// TIA Portal project "移位运算" (V13)

(* hardware
DEVICE "S7300/ET200M station_1"  S7-300 station
   slot 0: "导轨_0"  Rail  6ES7 390-1***0-0AA0
   slot 2: "PLC_1"  CPU 314C-2 PN/DP  6ES7 314-6EH04-0AB0  V3.3
      slot 2: "PROFINET 接口_1"  PN-IO
         slot 1: "Port_1"  Port
         slot 2: "Port_2"  Port
      slot 5: "DI 24/DO 16_1"  DI24/DO16
      slot 6: "AI 5/AO 2_1"  AI5/AO2
      slot 7: "计数_1"  Counter
      slot 8: "定位_1"  Positioning
*)

// ===== PLC "PLC_1"  CPU 314C-2 PN/DP =====

VAR_GLOBAL   // PLC tag table "默认变量表"
   "tag_1" AT %M0.0 : Bool;
   "tag_2" AT %M0.1 : Bool;
   "tag_3" AT %M0.2 : Bool;
   "tag_4" AT %MW100 : Int;
   "tag_5" AT %M0.3 : Bool;
   "tag_6" AT %M0.4 : Bool;
   "tag_7" AT %MW110 : Word;
   "tag_8" AT %MW120 : Word;
   "tag_9" AT %MW130 : Int;
END_VAR

ORGANIZATION_BLOCK "Main"   // OB1, LAD
TITLE = "Main Program Sweep (Cycle)"
{ S7_Optimized_Access := 'FALSE' }
VERSION : 0.1
   VAR_TEMP
      OB1_EV_CLASS : Byte;   // Bits 0-3 = 1 (Coming event), Bits 4-7 = 1 (Event class 1)
      OB1_SCAN_1 : Byte;   // 1 (Cold restart scan 1 of OB 1), 3 (Scan 2-n of OB 1)
      OB1_PRIORITY : Byte;   // Priority of OB Execution
      OB1_OB_NUMBR : Byte;   // 1 (Organization block 1, OB1)
      OB1_RESERVED_1 : Byte;   // Reserved for system
      OB1_RESERVED_2 : Byte;   // Reserved for system
      OB1_PREV_CYCLE : Int;   // Cycle time of previous OB1 scan (milliseconds)
      OB1_MIN_CYCLE : Int;   // Minimum cycle time of OB1 (milliseconds)
      OB1_MAX_CYCLE : Int;   // Maximum cycle time of OB1 (milliseconds)
      OB1_DATE_TIME : Date_And_Time;   // Date and time OB1 started
   END_VAR
BEGIN

REGION Network 1
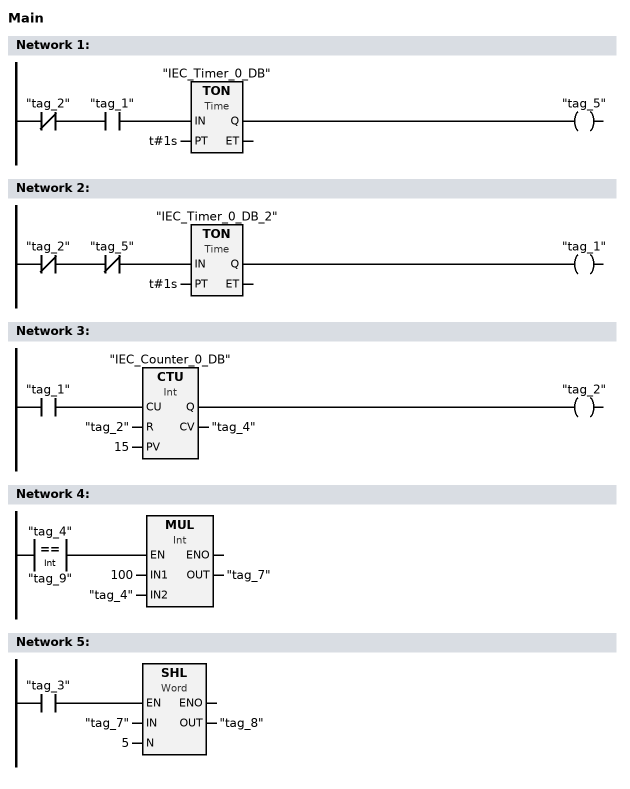
   "IEC_Timer_0_DB".TON(IN := NOT "tag_2" AND "tag_1", PT := t#1s);
   "tag_5" := "IEC_Timer_0_DB".Q;
END_REGION

REGION Network 2
   "IEC_Timer_0_DB_2".TON(IN := NOT "tag_2" AND NOT "tag_5", PT := t#1s);
   "tag_1" := "IEC_Timer_0_DB_2".Q;
END_REGION

REGION Network 3
   "IEC_Counter_0_DB".CTU(CU := "tag_1", R := "tag_2", PV := 15, CV => "tag_4");
   "tag_2" := "IEC_Counter_0_DB".Q;
END_REGION

REGION Network 4
   RUNG wire#powerrail
      { S7_Templates := "SrcType := Int" } EQ_Contact(in1 := "tag_4", in2 := "tag_9")
      { S7_Templates := "SrcType := Int"; S7_GenerateENO := "TRUE" } Mul(in1 := 100, in2 := "tag_4", out => "tag_7")
   END_RUNG
   // the same network as SCL:
   IF "tag_4" = "tag_9" THEN "tag_7" := 100 * "tag_4"; END_IF;
END_REGION

REGION Network 5
   RUNG wire#powerrail
      Contact( "tag_3" )
      { S7_Templates := "SrcType := Word"; S7_GenerateENO := "TRUE" } Shl(in := "tag_7", n := 5, out => "tag_8")
   END_RUNG
   // the same network as SCL:
   IF "tag_3" THEN "tag_8" := SHL(IN := "tag_7", N := 5); END_IF;
END_REGION
END_ORGANIZATION_BLOCK